TYPE ST_System_WP_Stellwert :
STRUCT
	Anford_SV_KW		: BOOL;
	Anford_SV_WW		: BOOL;
	Anford_WP			: BOOL;
END_STRUCT
END_TYPE

(* stored: Version 1.1.0.1, ProductVersion 3.1.4024.9
   DUT ST_System_WP_Stellwert: Id {d97d3600-684a-4709-93a7-444374d2ee21} *)
